FUNCTION_BLOCK COMPARE_5059E05E0748EACE (* Compare *)
  (* Standard: 61499-2 *)
  (* Version 1.1, 24.06.2019, winkhub, nxtControl GmbH, support all types *)
  PACKAGE UAO.Hackathon;
  (* Compiler Cpp *)
  {SET_ATTRIBUTE(Runtime.FBType.ImplementingType, Runtime.Standard#DYNGEN_COMPARE)}
  {SET_ATTRIBUTE(Configuration.GenericFBType.InterfaceParams, Runtime.Standard#CNT:=2;IN${CNT$}:STRING(255))}
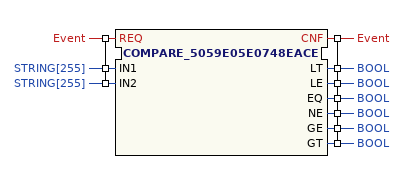
  EVENT_INPUT
    REQ WITH IN1, IN2; (* Normal Execution Request *)
  END_EVENT
  EVENT_OUTPUT
    CNF WITH LT, LE, EQ, NE, GE, GT; (* Execution Confirmation *)
  END_EVENT
  VAR_INPUT
    IN1 : STRING[255]; (* Argument *)
    IN2 : STRING[255]; (* Argument *)
  END_VAR
  VAR_OUTPUT
    LT : BOOL; (* IN1 < IN2 *)
    LE : BOOL; (* IN1 <= IN2 *)
    EQ : BOOL; (* IN1 = IN2 *)
    NE : BOOL; (* IN1 <> IN2 *)
    GE : BOOL; (* IN1 >= IN2 *)
    GT : BOOL; (* IN1 > IN2 *)
  END_VAR
  EC_STATES
    START;
  END_STATES
END_FUNCTION_BLOCK
